// SIMATIC S7-200 project (STEP 7-Micro/WIN), CPU 221 REL 01.10

SYMBOL_TABLE USER1
start            I0.0
estop2           I0.2
BT1              Q0.0
BT2              Q0.1
BT3              Q0.2
estop1           I0.1
END_SYMBOL_TABLE

ORGANIZATION_BLOCK MAIN:OB1
TITLE=PROGRAM COMMENTS
BEGIN
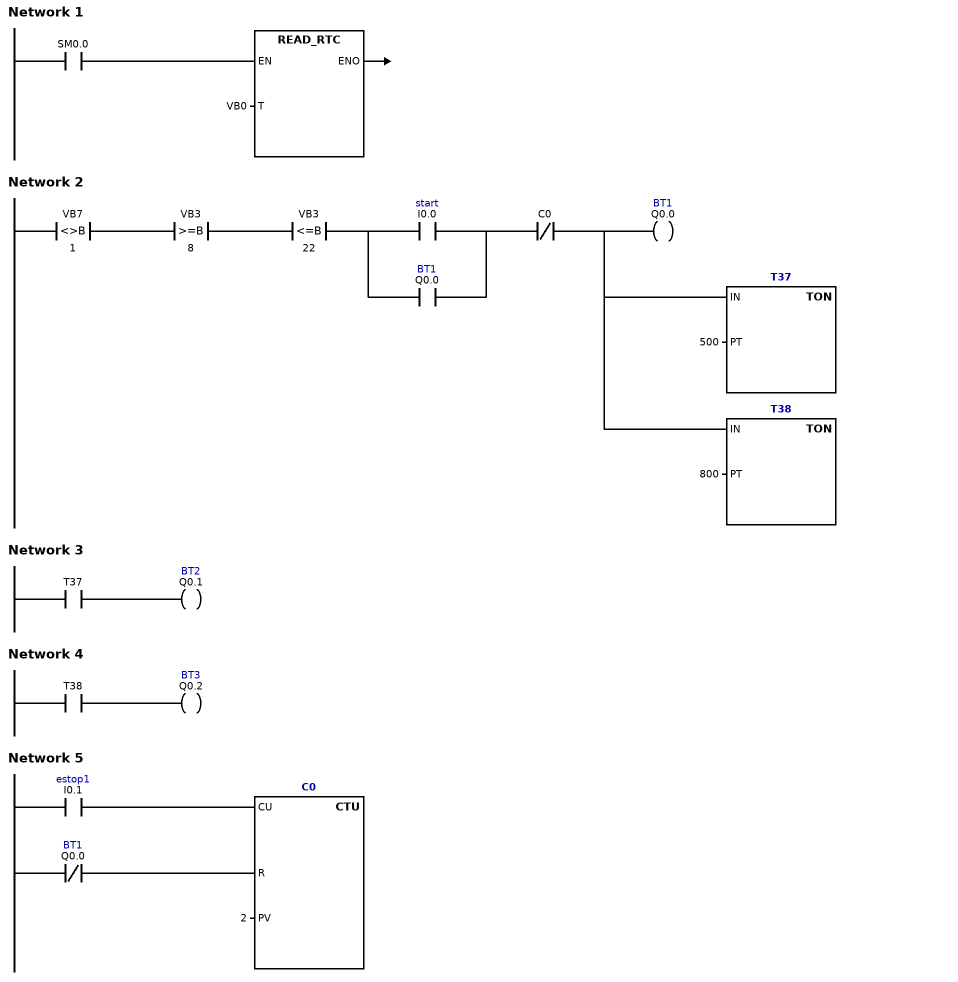
Network 1
LD     SM0.0
TODR   VB0
Network 2
// (network saved uncompiled; LAD cells follow)
// row 0: c0 -|<>B|- VB7, 1  c1 -|>=B|- VB3, 8  c2 -|<=B|- VB3, 22 v  c3 -| |- start:I0.0 v  c4 -|/|- C0 v  c5 -( ) BT1:Q0.0
// row 1: c2 ^  c3 -| |- BT1:Q0.0 ^  c4 ^v  c5 --  c6 [TON T37 IN:=power@row1, PT:=500]
// row 2: c4 ^v  c6 [box]
// row 3: c4 ^  c5 --  c6 [TON T38 IN:=power@row3, PT:=800]
// row 4: c6 [box]
Network 3
LD     T37
=      BT2:Q0.1
Network 4
LD     T38
=      BT3:Q0.2
Network 5
LD     estop1:I0.1
LDN    BT1:Q0.0
CTU    C0, 2
END_ORGANIZATION_BLOCK
